// TIA Portal V16 export
// export: Created 2024-08-29T13:26:37.0947873Z, ExportSetting WithDefaults, DisplayName Totally Integrated Automation Portal, DisplayVersion V16, DisplayName TIA Portal Version Control Interface, DisplayVersion V16, DisplayName TIA Portal Openness, DisplayVersion V16, DisplayName STEP 7 Professional, DisplayVersion V16, DisplayName STEP 7 Safety, DisplayVersion V16, DisplayName WinCC Professional, DisplayVersion V16
DATA_BLOCK "DB00802_St_ConstAqRawData"   // DB802
TITLE = Static DB [SYSTEM CONSTANTS] — Analog Input Card Types, Ranges and Parameters
{ S7_Optimized_Access := 'TRUE' }
AUTHOR : M_Gledhill
FAMILY : SysConstants
NAME : St_ConstAqRawData
VERSION : 1.0
// PRACTICAL SERIES AUTOMATION LIBRARY (PAL)   —   COPYRIGHT 2020 – M. GLEDHILL (MIT LICENCE)
//                   ———— ◆ ————
// FULL ONLINE DOCUMENTATION IS AVAILABLE AT: https://practicalseries.com/2001-pal/index.html
// stored: AutoNumber false, DBAccessibleFromOPCUA true, IsOnlyStoredInLoadMemory false, IsRetainMemResEnabled false, IsWriteProtectedInAS false, MemoryReserve 100
   VAR
      _DB_Header { ExternalAccessible := 'False'; ExternalVisible := 'False'; ExternalWritable := 'False'} : Array[0..79] of Bool;   // Static DB [SYSTEM CONSTANTS] — Analog Output Card Type, Range and Parameters
      __________0000_0 { ExternalAccessible := 'False'; ExternalVisible := 'False'; ExternalWritable := 'False'} : Bool := false;
      __________0000_1 { ExternalAccessible := 'False'; ExternalVisible := 'False'; ExternalWritable := 'False'} : Bool := false;
      revInfo { ExternalWritable := 'False'} : "UT01000_St_SysRevision";
      __________0010_0 { ExternalAccessible := 'False'; ExternalVisible := 'False'; ExternalWritable := 'False'} : Bool := false;
      __________0010_1 { ExternalAccessible := 'False'; ExternalVisible := 'False'; ExternalWritable := 'False'} : Bool := false;
      AQ_RAW_0000 { ExternalWritable := 'False'} : "UT00802_St_ConstAqRawData";   // AQ User defined signal type
      __________0020_0 { ExternalAccessible := 'False'; ExternalVisible := 'False'; ExternalWritable := 'False'} : Bool := false;
      __________0020_1 { ExternalAccessible := 'False'; ExternalVisible := 'False'; ExternalWritable := 'False'} : Bool := false;   // ▀▀▀▀ ANALOG INPUT SIGNAL — VOLTAGE
      AQ_RAW_1000 { ExternalWritable := 'False'} : "UT00802_St_ConstAqRawData";   // AQ Voltage (-10 V to +10 V)
      AQ_RAW_1001 { ExternalWritable := 'False'} : "UT00802_St_ConstAqRawData";   // AQ Voltage (-5 V to +5 V)
      AQ_RAW_1002 { ExternalWritable := 'False'} : "UT00802_St_ConstAqRawData";   // AQ Voltage (0 V to 10 V)
      AQ_RAW_1003 { ExternalWritable := 'False'} : "UT00802_St_ConstAqRawData";   // AQ Voltage (1 V to 5 V)
      __________0030_0 { ExternalAccessible := 'False'; ExternalVisible := 'False'; ExternalWritable := 'False'} : Bool;
      __________0030_1 { ExternalAccessible := 'False'; ExternalVisible := 'False'; ExternalWritable := 'False'} : Bool;   // ▀▀▀▀ ANALOG INPUT SIGNAL — CURRENT
      AQ_RAW_2000 { ExternalWritable := 'False'; S7_SetPoint := 'True'} : "UT00802_St_ConstAqRawData";   // AQ Current (-20 mA to +20 mA)
      AQ_RAW_2001 { ExternalWritable := 'False'; S7_SetPoint := 'True'} : "UT00802_St_ConstAqRawData";   // AQ Current (0 mA to 20 mA)
      AQ_RAW_2002 { ExternalWritable := 'False'; S7_SetPoint := 'True'} : "UT00802_St_ConstAqRawData";   // AQ Current (4 mA to 20 mA)
   END_VAR
BEGIN
   // _DB_Header[0] : ▄▄▄▄▄▄▄▄▄▄▄▄▄▄▄▄▄▄▄▄▄▄▄▄▄▄▄▄▄▄▄▄ ＣＯＮＳＴＡＮＴＳ ▄▄
   // _DB_Header[2] : TITLE: SYSTEM CONSTANTS — ANALOG OUTPUT CARD TYPE, RANGE AND PARAMETERS
   // _DB_Header[4] : ▀▀▀▀▀▀▀▀▀▀▀▀▀▀▀▀▀▀▀▀▀▀▀▀▀▀▀▀▀▀▀▀▀▀▀▀▀▀▀▀▀▀▀▀
   // _DB_Header[5] : TYPE: STATIC
   // _DB_Header[6] : ▄▄▄▄▄▄▄▄▄▄▄▄▄▄▄▄▄▄▄▄▄▄▄▄▄▄▄▄▄▄▄▄▄▄▄▄▄▄▄▄ ʷᴵᴰ⁻ᵈʰᵐ ▄
   // _DB_Header[8] : DB00802_St_ConstAqRawData is a static data block that holds a full set of range, parameter and
   // _DB_Header[9] : descriptive data for all types of analog output card channels.
   // _DB_Header[11] : Each dataset is stored in a structure of user data type: UT00802_St_ConstAqRawData. This structure
   // _DB_Header[12] : is configured to hold all the data required by the card itself, any module accessing an analog output
   // _DB_Header[13] : and any supervisory system that is to display the type and configuration of the output channel.
   // _DB_Header[15] : All the channel data is stored as constants and is used by all modules that have an interface
   // _DB_Header[16] : to an analog output card.
   // _DB_Header[18] : The purpose of the user data type and associated data block is to provide a consistent and
   // _DB_Header[19] : tested set of range, parameter and descriptive data that can be used directly by modules that
   // _DB_Header[20] : interface with analog output cards.
   // _DB_Header[22] : The ranges correspond to the numerical values required by the card for a given type of analog card
   // _DB_Header[23] : signal. For example, a 4-20 mA card requires a numerical value of 0 to generate an output of
   // _DB_Header[24] : 4 mA ranging up to a value of 27648 at 20 mA. The data specified in the UT00802 variable would
   // _DB_Header[25] : have a lower limit of 0 and an upper limit of 27648.
   // _DB_Header[27] : In addition, each dataset contains the parametric data that defines the particular channel type and
   // _DB_Header[28] : can be used to set a particular analog output channel to a particular type and range during
   // _DB_Header[29] : runtime. Each dataset also contains a textual description of the channel type,
   // _DB_Header[30] : e.g. Current (4 mA to 20 mA)
   // _DB_Header[31] : for display and information purposes.
   // _DB_Header[33] : The PDF version of the SMDS for this module is avAQlable online here:
   // _DB_Header[34] : http://psop.uk/pal-smds-db00802-p
   // _DB_Header[36] : ━━━ ⬙⬙⬙⬙⬙⬙ ━━━
   // _DB_Header[38] : ▄▄▄▄▄▄▄▄▄▄▄▄▄▄▄▄▄▄▄▄▄▄▄▄▄▄▄▄▄▄▄▄▄▄▄▄▄▄▄▄▄▄▄▄
   // _DB_Header[39] : MODIFICATION HISTORY
   // _DB_Header[41] : This is a summary of the recent software modifications made to this block (most recent at top)
   // _DB_Header[43] : ―――――――――――――――――――――――――――――――――――――――――――
   // _DB_Header[44] : DATE REVISION MASTER BRANCH DEV
   // _DB_Header[45] : (nnn.amm) COMMIT TAG (Base ---> Merge) BRANCH Author
   // _DB_Header[46] : ———————————————————————————————————————————
   // _DB_Header[47] : 2024.05.17 001.000 D0017A-000.106 D0017 N/A D0017A M. Gledhill
   // _DB_Header[48] : DB00802 Block created
   // _DB_Header[49] : ———————————————————————————————————————————
   // _DB_Header[50] : Where: nnn = Major revision
   // _DB_Header[51] : a = Type (1-7 Development, 8 Proving, 9 Qualification, 0 Release)
   // _DB_Header[52] : mm = Minor revision (must be 00 if a = 0)
   // _DB_Header[53] : Block properties version number should be set to nn.a (only one decimal place)
   // _DB_Header[55] : ██████████████ █ █ █ █ END █ █ █ █ ██████████████
   revInfo.REV_BLOCK := 'DB00802';
   revInfo.REV_NUMBER := '001.000';
   revInfo.REV_DATE := '2024-05-17';
   revInfo.REV_AUTHOR := 'M. Gledhill';
   // AQ_RAW_0000.RAW_DESC : Signal type description (plAQn English)
   AQ_RAW_1000.AQ_CODE := 16#1000;
   AQ_RAW_1000.RAW_MIN := -27648;
   AQ_RAW_1000.RAW_MAX := 27648;
   AQ_RAW_1000.RAW_DESC := 'Voltage (-10 V to +10 V)';   // Signal type description (plAQn English)
   AQ_RAW_1000.PARAM_TYPE := 16#01;
   AQ_RAW_1000.PARAM_RANGE := 16#00;
   AQ_RAW_1001.AQ_CODE := 16#1001;
   AQ_RAW_1001.RAW_MIN := -27648;
   AQ_RAW_1001.RAW_MAX := 27648;
   AQ_RAW_1001.RAW_DESC := 'Voltage (-5 V to +5 V)';   // Signal type description (plAQn English)
   AQ_RAW_1001.PARAM_TYPE := 16#01;
   AQ_RAW_1001.PARAM_RANGE := 16#01;
   AQ_RAW_1002.AQ_CODE := 16#1002;
   AQ_RAW_1002.RAW_MIN := 0;
   AQ_RAW_1002.RAW_MAX := 27648;
   AQ_RAW_1002.RAW_DESC := 'Voltage (0 V to 10 V)';   // Signal type description (plAQn English)
   AQ_RAW_1002.PARAM_TYPE := 16#01;
   AQ_RAW_1002.PARAM_RANGE := 16#02;
   AQ_RAW_1003.AQ_CODE := 16#1003;
   AQ_RAW_1003.RAW_MIN := 0;
   AQ_RAW_1003.RAW_MAX := 27648;
   AQ_RAW_1003.RAW_DESC := 'Voltage (1 V to 5 V)';   // Signal type description (plAQn English)
   AQ_RAW_1003.PARAM_TYPE := 16#01;
   AQ_RAW_1003.PARAM_RANGE := 16#03;
   AQ_RAW_2000.AQ_CODE := 16#2000;
   AQ_RAW_2000.RAW_MIN := -27648;
   AQ_RAW_2000.RAW_MAX := 27648;
   AQ_RAW_2000.RAW_DESC := 'Current (-20 mA to +20 mA)';
   AQ_RAW_2000.PARAM_TYPE := 16#02;
   AQ_RAW_2000.PARAM_RANGE := 16#00;
   AQ_RAW_2001.AQ_CODE := 16#2001;
   AQ_RAW_2001.RAW_MIN := 0;
   AQ_RAW_2001.RAW_MAX := 27648;
   AQ_RAW_2001.RAW_DESC := 'Current (0 mA to 20 mA)';
   AQ_RAW_2001.PARAM_TYPE := 16#02;
   AQ_RAW_2001.PARAM_RANGE := 16#01;
   AQ_RAW_2002.AQ_CODE := 16#2002;
   AQ_RAW_2002.___________0020_0 := false;
   AQ_RAW_2002.___________0020_1 := false;
   AQ_RAW_2002.RAW_MIN := 0;
   AQ_RAW_2002.RAW_MAX := 27648;
   AQ_RAW_2002.RAW_DESC := 'Current (4 mA to 20 mA)';
   AQ_RAW_2002.PARAM_TYPE := 16#02;
   AQ_RAW_2002.PARAM_RANGE := 16#02;
END_DATA_BLOCK
